FUNCTION_BLOCK Publisher (* Template for an empty simple function block *)
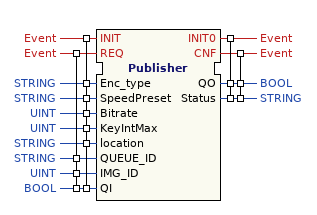
  EVENT_INPUT
    INIT WITH Enc_type, SpeedPreset, location, KeyIntMax, Bitrate, QI;
    REQ WITH QUEUE_ID, IMG_ID, QI; (* Normal Execution Request *)
  END_EVENT
  EVENT_OUTPUT
    INIT0 WITH QO, Status;
    CNF WITH QO, Status; (* Execution Confirmation *)
  END_EVENT
  VAR_INPUT
    Enc_type : STRING;
    SpeedPreset : STRING;
    Bitrate : UINT;
    KeyIntMax : UINT;
    location : STRING;
    QUEUE_ID : STRING;
    IMG_ID : UINT;
    QI : BOOL;
  END_VAR
  VAR_OUTPUT
    QO : BOOL;
    Status : STRING;
  END_VAR
END_FUNCTION_BLOCK
